Staubli VAL3: refreshExport.pgx

program refreshExport(bool x_bShowLine (dimensions=1), string x_sPath (dimensions=1))
  local num l_nLocal
  local string l_sEmpty
  local string l_sItem
begin
  call use:setSizeList(19,0,19,11)
  call use:listcreate("ROBOT")
  call use:stringCopy(l_sEmpty,sExport)
  call use:listempty()
  //
  // build the list
  if libList(x_sPath,sExport)
    // build and refresh
    if x_sPath!="Disk://../"
      l_sItem=".."
      call use:listadd(l_sItem)
    endIf
    call use:listadd(sExport)
    use:nView=nView
    call use:listredraw(nIndex-nView)
    if !x_bShowLine
      call use:listcursor(nView,false)
    endIf
  endIf
end
